RoboDK station: Custom_Social_Task.rdk

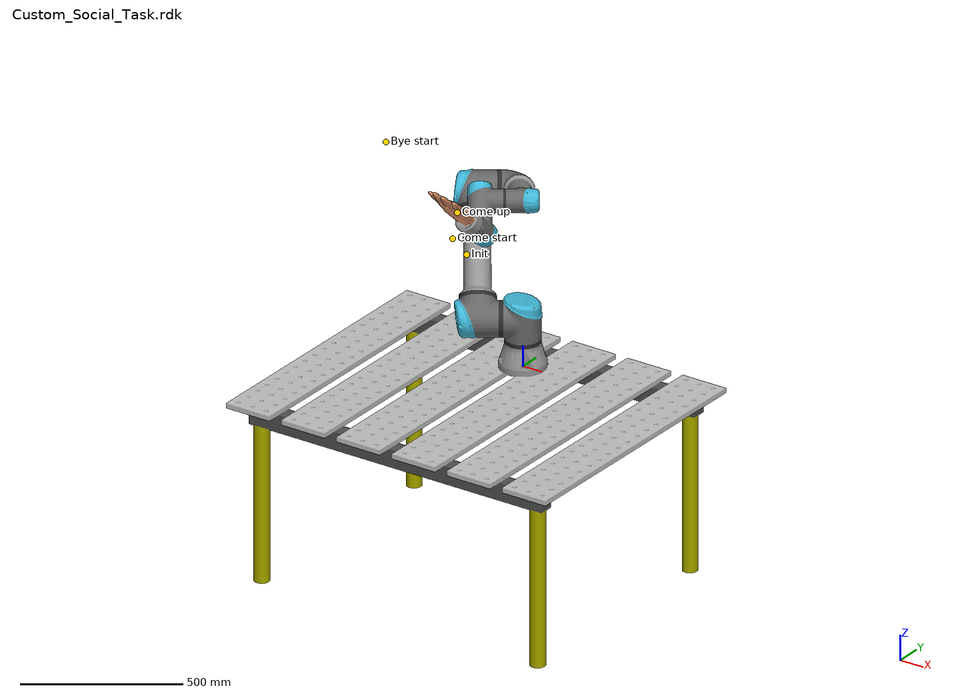
[picture v0: the station drawn from its stored meshes, robots at their saved joint values, targets as dots, program paths as lines]
Station Assistive_UR5e_SW (saved by RoboDK 5.9.2). Poses are relative to the parent item; angles as X-Y-Z fixed-axis rotations.
  - frame UR5e Base at (0, 0, 0) mm
    - robot UR5e: 6 axes, payload 5 kg, reach 850 mm, repeatability 0.03 mm, weight 18.4 kg
        modified DH rows (alpha deg, a mm, theta deg, d mm): 0, 0, 0, 162.5; 90, 0, 180, 0; 0, 425, 0, 0; 0, 392.25, 0, 133.3; -90, 0, 0, 99.7; 90, 0, 180, 99.6
        joint limits [-360, -360, -360, -360, -360, -360] to [360, 360, 360, 360, 360, 360]; home [0, -90, -90, 0, 90, 0]; saved at [-54.185, -44.005, -115.567, 210.121, -61.689, 234.556]
      - tool Hand, TCP at (0, 0, 50) mm, size 54.8 x 155.9 x 193.5 mm, geometry from Hand.stl
  - frame World at (0, 0, 0) mm
    - object Table at (0, 0, 0) mm, size 1193.8 x 965.2 x 609.6 mm, geometry from welding_table.sld
    - target Init (joint target) at (0, -300, 500) mm, rotated rx 90 ry 0 rz 0 deg; joints [-27.588, -45.348, -114.543, 159.891, -27.588, 0] of UR5e
    - target Hello start (joint target) at (0, -300, 500) mm, rotated rx 0 ry 0 rz 90 deg; joints [-63.619, -66.936, -144.253, 301.188, -90, 63.619] of UR5e
    - target Hello left (joint target) at (0, -300, 500) mm, rotated rx -31.9 ry 0.01 rz 90.02 deg; joints [-49.788, -72.342, -143.856, 328.09, -66.193, 45.138] of UR5e
    - target Hello right (joint target) at (0, -300, 500) mm, rotated rx 42.12 ry 0 rz 90.02 deg; joints [-83.57, -65.793, -136.862, 286.894, -131.794, 81.384] of UR5e
    - target Bye start (joint target) at (-300, -300, 800) mm, rotated rx 0 ry 0 rz 90 deg; joints [-116.688, -78.781, -90.787, 259.568, -90, 116.688] of UR5e
    - target Bye left (joint target) at (-300, -300, 800) mm, rotated rx 0 ry 0 rz 45 deg; joints [-116.688, -78.781, -90.787, 259.568, -90, 71.688] of UR5e
    - target Bye right (joint target) at (-300, -300, 800) mm, rotated rx 0 ry 0 rz 135 deg; joints [-116.688, -78.781, -90.787, 259.568, -90, 161.688] of UR5e
    - target Come start (joint target) at (-51.45, -300, 539.1) mm, rotated rx 87.76 ry 83.31 rz -10.42 deg; joints [-41.832, -48.545, -107.847, 156.862, -33.639, 276.29] of UR5e
    - target Come up (joint target) at (-35.39, -300, 633.01) mm, rotated rx -5.89 ry 46.89 rz -102.52 deg; joints [-54.185, -44.005, -115.567, 210.121, -61.689, 234.556] of UR5e
